INTERFACE IF_queueManager

PROPERTY currentLevel : INT(1..NUMLEVELS)
SET
END_SET
END_PROPERTY

METHOD doneAck
VAR_INPUT
END_VAR
END_METHOD

PROPERTY queue : REFERENCE TO ARRAY [1..NUMLEVELS] OF INT
GET
END_GET
END_PROPERTY

METHOD reset
VAR_INPUT
END_VAR
END_METHOD

END_INTERFACE

(* stored: Version 1.1.0.1, ProductVersion 3.1.4024.6
   Itf IF_queueManager: Id {0614bf0d-28f4-4560-b0fe-dc1c17c4dea8}
   Property currentLevel: Id {6ba6c7c2-b083-4143-91e8-0ad03a37d3e2}
   Set Set: Id {1769bcef-77f7-4d76-b4eb-8f91f920bd1d}
   Method doneAck: Id {5a2bb297-cc5a-4c29-9a61-2f9dbe0a0fab}
   Property queue: Id {99997325-aa61-4eb8-b341-38be5307f03c}
   Get Get: Id {9748c0d4-e1b0-48a7-932f-57b67b0e0795}
   Method reset: Id {f08d815b-2869-4435-b30e-50a5683fb81f} *)
